FUNCTION_BLOCK Test_F_TimeAsString_ms_ReturnsTimeString_ms EXTENDS TUnitTestBase
VAR
    TimeStruct : TIMESTRUCT := (wHour := 6, wMinute := 5, wSecond := 4, wMilliseconds := 135);
END_VAR

Assertion.AssertEquals_STRING(
    Expected := '06:05:04.135',
    Actual   := F_TimeAsString_ms(TimeStruct),
    ObjectName := _TestName,
    VariableName  := 'F_TimeAsString_ms(TimeStruct)');


TestFinished();

END_FUNCTION_BLOCK

(* stored: Version 1.1.0.1, ProductVersion 3.1.4024.4
   POU Test_F_TimeAsString_ms_ReturnsTimeString_ms: Id {cfe81a32-3eca-0666-0352-ea68d5a05067}, SpecialFunc None *)
